FUNCTION_BLOCK D_5States_1Algo (* Basic FB with empty ECC *)
  (* Standard: 61499-2 *)
  (* Version 1.0, 2023-09-22, AK124910 *)
  PACKAGE servSeq;
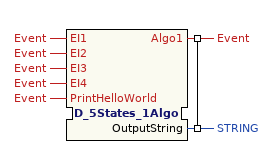
  EVENT_INPUT
    EI1;
    EI2;
    EI3;
    EI4;
    PrintHelloWorld;
  END_EVENT
  EVENT_OUTPUT
    Algo1 WITH OutputString;
  END_EVENT
  VAR_OUTPUT
    OutputString : STRING;
  END_VAR
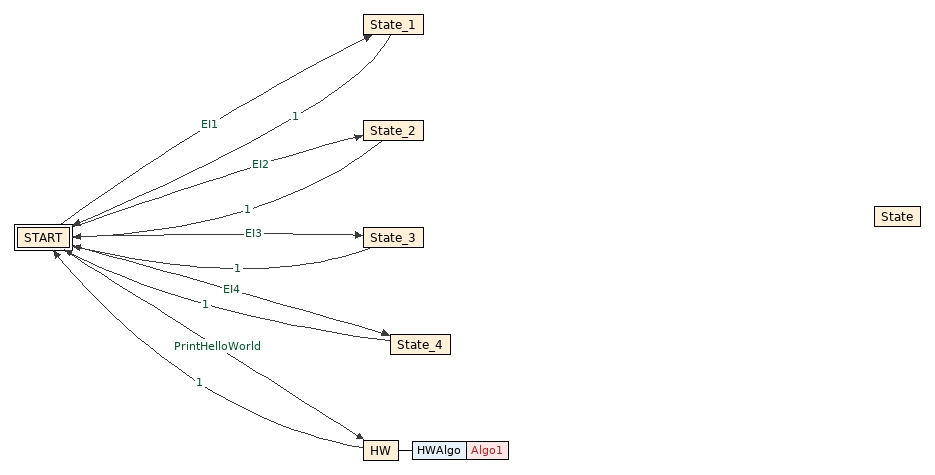
  EC_STATES
    START; (* Initial State *)
    State_1;
    State_2;
    State_3;
    HW : HWAlgo -> Algo1;
    State;
    State_4;
  END_STATES
  EC_TRANSITIONS
    START TO State_1 := EI1;
    State_1 TO START := 1;
    START TO State_2 := EI2;
    State_2 TO START := 1;
    START TO State_3 := EI3;
    State_3 TO START := 1;
    START TO State_4 := EI4;
    State_4 TO START := 1;
    START TO HW := PrintHelloWorld;
    HW TO START := 1;
  END_TRANSITIONS
  ALGORITHM HWAlgo IN ST:
OutputString := CONCAT(OutputString, 'H');
OutputString := CONCAT(OutputString, 'E');
OutputString := CONCAT(OutputString, 'L');
OutputString := CONCAT(OutputString, 'L');
OutputString := CONCAT(OutputString, 'O');
OutputString := CONCAT(OutputString, ' ');
OutputString := CONCAT(OutputString, 'W');
OutputString := CONCAT(OutputString, 'O');
OutputString := CONCAT(OutputString, 'R');
OutputString := CONCAT(OutputString, 'L');
OutputString := CONCAT(OutputString, 'D');
OutputString := CONCAT(OutputString, '!');
  END_ALGORITHM
  SERVICE external/internal_interface (* Basic FB with empty ECC *)
    SEQUENCE ServiceSequence (* Coverage: 1.0 *) {SET_ATTRIBUTE(StartState, START)}
      external.EI1();
      external.EI2();
      external.EI3();
      external.EI4();
      external.PrintHelloWorld() -> external.Algo1(OutputString:=STRING#'HELLO WORLD!';);
    END_SEQUENCE
    SEQUENCE ServiceSequence2 (* Coverage: 1.0 *) {SET_ATTRIBUTE(StartState, START)}
      external.PrintHelloWorld() -> external.Algo1(OutputString:=STRING#'HELLO WORLD!';);
      external.EI1();
      external.EI2();
      external.EI3();
      external.EI4();
    END_SEQUENCE
  END_SERVICE
END_FUNCTION_BLOCK
